{attribute 'GeneratedUsingTerminal: EL6201-0000-0017'}
{attribute addProperty BoxType "EL6201-0000-0017"}
{attribute addProperty Id "Slave_17A_DI0BOOL1Slave_17A_DI1BOOL1Slave_17A_DI2BOOL1Slave_17A_DI3BOOL1Slave_17B_DI0BOOL1Slave_17B_DI1BOOL1Slave_17B_DI2BOOL1Slave_17B_DI3BOOL1"}
{attribute addProperty CRC "848952453"}
{attribute addProperty Size "8"}
TYPE Slave_17_Inputs_3299FC85 :
STRUCT
	{attribute addProperty Name "Slave_17A_DI0"}
	Slave_17A_DI0 : BOOL;
	{attribute addProperty Name "Slave_17A_DI1"}
	Slave_17A_DI1 : BOOL;
	{attribute addProperty Name "Slave_17A_DI2"}
	Slave_17A_DI2 : BOOL;
	{attribute addProperty Name "Slave_17A_DI3"}
	Slave_17A_DI3 : BOOL;
	{attribute addProperty Name "Slave_17B_DI0"}
	Slave_17B_DI0 : BOOL;
	{attribute addProperty Name "Slave_17B_DI1"}
	Slave_17B_DI1 : BOOL;
	{attribute addProperty Name "Slave_17B_DI2"}
	Slave_17B_DI2 : BOOL;
	{attribute addProperty Name "Slave_17B_DI3"}
	Slave_17B_DI3 : BOOL;
END_STRUCT
END_TYPE

(* stored: Version 1.2.0.0, ProductVersion 3.1.4024.9
   DUT Slave_17_Inputs_3299FC85: Id {caedcf42-8c65-437d-88bc-d679cdaa4446} *)
